// TIA Portal V20 export
TYPE "typeCmControlNodeBrakeTest"
// stored: Namespace Unit1.Em13
   STRUCT
      jrUnIoadingPnPAxisZ : "LER_typeBrakeTestEmControlNodes";
   END_STRUCT;
END_TYPE
